TYPE ST_MasterAxisPos :
STRUCT
	Pos		: DINT:=0;
	PosLast 	: DINT:=0;
END_STRUCT
END_TYPE

(* stored: Version 1.1.0.1, ProductVersion 3.1.4024.9
   DUT ST_MasterAxisPos: Id {028035cd-8ec1-4908-ab50-02c2e817306f} *)
